FUNCTION_BLOCK EL3208
VAR
	_io : EL3xx8_Data;
	{attribute addProperty Name "WcState"}
	_wcState : WcStateInputToggle;
	{attribute addProperty Name "Info data"}
	_infoData : InfoDataAds;
END_VAR

PROPERTY IO : REFERENCE TO EL3xx8_Data
GET
IO REF= _io;
END_GET
END_PROPERTY

PROPERTY WcState : REFERENCE TO WcStateInputToggle
GET
WcState REF= _wcState;
END_GET
END_PROPERTY

END_FUNCTION_BLOCK

(* stored: Version 1.1.0.1, ProductVersion 3.1.4024.9
   POU EL3208: Id {4be725e5-0b4e-0a0f-21ad-4778ce8d2b6e}, SpecialFunc None
   Property IO: Id {511aca9a-5d98-0320-15eb-94608decd7cf}
   Get Get: Id {eb44f308-3189-0a4b-2778-34ed060107b9}
   Property WcState: Id {ddb08bb4-4d31-0929-0709-cad73f110499}
   Get Get: Id {9359325e-35c8-0bce-2884-4675475dca7a} *)
